// TwinCAT 3 PLC project Potentiometer_Inlezen
// ProgramVersion: 3.1.4024.0
// libraries:
//   Tc2_Standard, * (Beckhoff Automation GmbH)
//   Tc2_System, * (Beckhoff Automation GmbH)
//   Tc3_Module, * (Beckhoff Automation GmbH)
// project tree:
//   / PlcTask.TcTTO
//   POUs/ MAIN.TcPOU
// real-time tasks:
//   TASK PlcTask: cycle T#10ms, priority 20, ADS port 350
//   TASK PlcTask1: cycle T#10ms, priority 21, ADS port 351
//   TASK PlcTask2: cycle T#10ms, priority 22, ADS port 352
//   TASK PlcTask3: cycle T#10ms, priority 26, ADS port 353
//   TASK PlcTask4: cycle T#10ms, priority 25, ADS port 354
//   TASK PlcTask5: cycle T#10ms, priority 24, ADS port 355
//   TASK PlcTask6: cycle T#10ms, priority 23, ADS port 356
//   TASK PlcTask7: cycle T#10ms, priority 27, ADS port 357

CONFIGURATION Potentiometer_Inlezen
    RESOURCE PLC ON TwinCAT3
        TASK PlcTask(INTERVAL := T#10ms, PRIORITY := 20);
        PROGRAM MAIN WITH PlcTask : MAIN;
    END_RESOURCE
END_CONFIGURATION

// ---- POUs/MAIN.TcPOU
PROGRAM MAIN
VAR
	Waarde: BYTE;
	potentiometer: INT;
END_VAR

(*
Potentiometer inlezen (maximaal 1 regels)

Lees de potentiometer in en verschaal deze waarden naar een getal tussen 0 en 100.
*)
Waarde:=LREAL_TO_BYTE(100*(potentiometer/32767.0));

END_PROGRAM
